Fanuc KAREL source: kt00081.KL

-- PROVISIONAL review KL for V1013-1; original PC SHA256 3932a47f35acd455cbfb859e4e9f9dc3692d7edd596ae8e1c0318e4e8383dcea
-- Incomplete behavior may be omitted. Consult companion uncertainty JSON. Do not deploy.
PROGRAM KT00081
%NOLOCKGROUP
VAR
  I2 : INTEGER
  OUT : INTEGER
-- UNRESOLVED_DECL Y1 type=002018
BEGIN
  -- UNRESOLVED_PC offsets 5-19; opcodes 2E,22,9D,33,B2
  -- UNRESOLVED_PC offsets 24-35; opcodes 2E,23
  -- UNRESOLVED_PC offsets 40-62; opcodes 22,9D,33,B1,21,54,23
  -- UNRESOLVED_PC offsets 67-71; opcodes 7F
END KT00081
